TYPE ST_ProcessVariables :
STRUCT
	fPower:REAL;
	fFlowSpeed:REAL;
	fGeneratorSpeed:REAL;
	fPitchAngle:REAL;
END_STRUCT
END_TYPE

(* stored: Version 1.1.0.1, ProductVersion 3.1.4024.9
   DUT ST_ProcessVariables: Id {6edc143a-675a-42a1-8ce3-6bb10f3702b9} *)
